// TIA Portal project "auto_level_palletizer_with_rotating_platform" (V15)

(* hardware
DEVICE "S7300/ET200M station_1"  S7-300 station
   slot 0: "Rail_0"  Rail  6ES7 390-1***0-0AA0
   slot 2: "controller_ALPwRP_system"  CPU 314C-2 PN/DP  6ES7 314-6EH04-0AB0  V3.3
      slot 2: "PROFINET interface_1"  PN-IO
         slot 1: "Port_1"  Port
         slot 2: "Port_2"  Port
      slot 5: "DI 24/DO 16_1"  DI24/DO16
      slot 6: "AI 5/AO 2_1"  AI5/AO2
      slot 7: "Count_1"  Counter
      slot 8: "Positioning_1"  Positioning
DEVICE "SINAMICS G_1"  Sinamics.Device
   slot 0: "CU240E-2 PN-F"  G120 CU240E-2 PN-F  6SL3244-0BB13-1FA0  4.7.9
      slot 1: "PROFINET interface"  MDD-SinamicsG120-P
   slot 0: "	_0"  Rail  SinamicsG120RackPN
   slot 3: "PM340 IP20"  PM340 IP20  6SL3210-1SB11-0AA0  -
*)

// ===== PLC "controller_ALPwRP_system"  CPU 314C-2 PN/DP =====

VAR_GLOBAL   // PLC tag table "Default tag table"
   "1B1" AT %I0.0 : Bool;   // Carton Passed
   "2B1" AT %I0.1 : Bool;   // Carton Counter
   "3B1" AT %I0.2 : Bool;   // Feeding Actuator 3A Fully Retracted
   "3B2" AT %I0.3 : Bool;   // Feeding Actuator 3A Fully Extended
   "3B3" AT %I0.4 : Bool;   // Feeding Actuator 3A in X position
   "4B1" AT %I0.5 : Bool;   // Sheet Motor 4A Fully Retracted
   "4B2" AT %I0.6 : Bool;   // Sheet Motor 4A Fully Extended
   "4B3" AT %I0.7 : Bool;   // Sheet Motor 4A in L position
   "5B1" AT %I1.0 : Bool;   // Carton to the feeding station
   "6B1" AT %I1.1 : Bool;   // Rotating Platform is ready (90 degrees)
   "7B1" AT %I1.2 : Bool;   // Hydraulic lift 6A Fully extended
   "7B2" AT %I1.3 : Bool;   // Hydraulic lift 6A Fully retracted
   "7B3" AT %I1.4 : Bool;   // Hydrauic Cylinder in Y
   "8B1" AT %I1.5 : Bool;   // Pallet Available
   "9B1" AT %I1.6 : Bool;   // Alignment Stopper 7A Fully Extended
   "9B2" AT %I1.7 : Bool;   // Alignment Stopper 7A Fully Retracted
   "10B1" AT %I2.0 : Bool;   // Carton to Alignment Actuator
   "S1" AT %I2.1 : Bool;   // START BUTTON PUSHED
   "S2" AT %I2.2 : Bool;   // STOP BUTTON PUSHED
   "S3" AT %I2.3 : Bool;   // RESET BUTTON PUSHED
   "EM_STOP" AT %I2.4 : Bool;   // EMERGENCY BUTTON PUSHED
   "11B1" AT %I2.5 : Bool;   // 8 AWG Carton Type
   "11B2" AT %I2.6 : Bool;   // 10 AWG Carton Type
   "11B3" AT %I2.7 : Bool;   // 12, 14, & 16 AWG Carton Types
   "M1" AT %Q0.0 : Bool;   // Belt Conveyor 1A
   "M2" AT %Q0.1 : Bool;   // Roller Conveyor 2A
   "M3" AT %Q0.2 : Bool;   // Feeding Actuator 3A
   "M4" AT %Q0.3 : Bool;   // Sheet Metal
   "P2" AT %Q0.4 : Bool;   // Pallet Rotation 5A
   "P1" AT %Q0.5 : Bool;   // Pallet z Axis 6A
   "A2" AT %Q0.6 : Bool;   // Aligment Stopper 7A
   "Tag_1" AT %M0.0 : Bool;
END_VAR

DATA_BLOCK "Main Program_DB"   // DB2
{ S7_Optimized_Access := 'FALSE' }
VERSION : 0.1
// stored: InstanceOfName Main Program
"Main Program"
BEGIN
END_DATA_BLOCK

FUNCTION_BLOCK "Main Program"   // FB1, GRAPH
{ S7_Optimized_Access := 'FALSE' }
VERSION : 0.1
   VAR_INPUT
      OFF_SQ : Bool := false;   // Turn sequence off
      INIT_SQ : Bool := false;   // Set sequence to initial state
      ACK_EF : Bool := false;   // Acknowledge all errors and faults
      S_PREV : Bool := false;   // Output previous step in parameter S_NO
      S_NEXT : Bool := false;   // Indicate next step in parameter S_NO
      SW_AUTO : Bool := false;   // Automatic mode
      SW_TAP : Bool := false;   // Semiautomatic/switch with transition
      SW_TOP : Bool := false;   // Semiautomatic/ignore transition
      SW_MAN : Bool := false;   // Manual mode
      S_SEL : Int := 0;   // Select step to be output to S_NO
      S_ON : Bool := false;   // Activate step indicated in S_NO
      S_OFF : Bool := false;   // Deactivate step indicated S_NO
      T_PUSH : Bool := false;   // Enable transition to switch in semi automatic mode
   END_VAR
   VAR_OUTPUT
      S_NO : Int := 0;   // Step number
      S_MORE : Bool := false;   // More steps are available and can be shown in S_NO
      S_ACTIVE : Bool := false;   // Step indicated in S_NO is active
      ERR_FLT : Bool := false;   // Interlock or supervision group error
      AUTO_ON : Bool := false;   // Automatic mode is active
      TAP_ON : Bool := false;   // Semiautomatic mode/step with transition enabled
      TOP_ON : Bool := false;   // Semiautomatic mode/ignore transition enabled
      MAN_ON : Bool := false;   // Manual mode is active
   END_VAR
   VAR
      in_initial_position : Bool;
      SWITCH : Array[0..0] of DWord;
      SW_SQTS : Array[0..21] of Byte;
      SW_ADDR : Word := 16#C;
      G7T_0 : GraphTransition;
      G7S_0 : GraphStep;
      PRE_CRIT : Array[0..0] of DWord;
      POST_CRIT : Array[0..0] of DWord;
      TVX : Array[0..5] of Byte;
      TTX : Array[0..5] of Byte;
      TSX : Array[0..2] of Byte;
      S00X : Array[0..2] of Byte;
      SOFFX : Array[0..2] of Byte;
      SONX : Array[0..2] of Byte;
      SAX : Array[0..2] of Byte;
      SERRX : Array[0..22] of Byte;
      SMX : Array[0..22] of Byte;
      S0X : Array[0..22] of Byte;
      S1X : Array[0..22] of Byte;
      S_DISPLAY : Int;   // Internal display of output parameter S_NO
      S_SEL_OLD : Int;   // Previous value in S_SEL
      S_DISPIDX : Byte;   // Index of the step in S_NO
      T_DISPIDX : Byte;   // Index of the transition displayed in T_NO
      MOPEDGE : Struct
         AUTO : Bool := false;
         MAN : Bool := false;
         TAP : Bool := false;
         TOP : Bool := false;
         ACK_S : Bool := false;
         REG_S : Bool := false;
         T_PREV : Bool := false;
         T_NEXT : Bool := false;
         LOCK : Bool := false;
         SUP : Bool := false;
         ACKREQ : Bool := false;
         SSKIP : Bool := false;
         OFF : Bool := false;
         INIT : Bool := false;
         HALT : Bool := false;
         TMS_HALT : Bool := false;
         OPS_ZERO : Bool := false;
         SACT_DISP : Bool := false;
         SEF_DISP : Bool := false;
         SALL_DISP : Bool := false;
         S_PREV : Bool := false;
         S_NEXT : Bool := false;
         S_SELOK : Bool := false;
         S_ON : Bool := false;
         S_OFF : Bool := false;
         T_PUSH : Bool := false;
         REG : Bool := false;
         ACK : Bool := false;
         IL_PERM : Bool := false;
         T_PERM : Bool := false;
         ILP_MAN : Bool := false;
      END_STRUCT;
      MOP : Struct   // Mode
         AUTO : Bool := true;   // Status: automatic mode
         MAN : Bool := false;   // Status: manual mode
         TAP : Bool := false;   // Status: semi automatic/switch with transition
         TOP : Bool := false;   // Status: semi automatic/ignore transition
         ACK_S : Bool := false;   // Request: acknowledge step at parameter S_NO
         REG_S : Bool := false;   // Request: register step indicated in S_NO
         T_PREV : Bool := false;   // Request: output previous valid transition in T_NO
         T_NEXT : Bool := false;   // Request: output next valid transition in T_NO
         LOCK : Bool := true;   // Status: interlocks activated
         SUP : Bool := true;   // Status: supervisions activated
         ACKREQ : Bool := true;   // Status: acknowledgment required
         SSKIP : Bool := false;   // Status: "Skip steps" enabled
         OFF : Bool := false;   // Request: deactivate all steps
         INIT : Bool := true;   // Request: set sequence to initial state
         HALT : Bool := false;   // Status: sequence halted
         TMS_HALT : Bool := false;   // Status: all internal timers held
         OPS_ZERO : Bool := false;   // Status: set all operands processed with N, L, D instructions to 0
         SACT_DISP : Bool := true;   // Status: display active steps only
         SEF_DISP : Bool := false;   // Status: display only steps with errors and disrupted steps
         SALL_DISP : Bool := false;   // Status: display all steps
         S_PREV : Bool := false;   // Request: output previous step to S_NO
         S_NEXT : Bool := false;   // Request: Output next step at S_NO parameter
         S_SELOK : Bool := false;   // Request: output step number from S_SEL to S_NO
         S_ON : Bool := false;   // Request: activate step indicated in S_NO
         S_OFF : Bool := false;   // Request: deactivate step at parameter S_NO
         T_PUSH : Bool := false;   // Request: transition switching enabled
         REG : Bool := false;   // Request: register all interlock and supervision errors
         ACK : Bool := false;   // Request: acknowledge all interlock and supervision errors
         IL_PERM : Bool := false;   // Status: permanent processing of all interlocks
         T_PERM : Bool := false;   // Status: permanent processing of all transitions
         ILP_MAN : Bool := false;   // Status: permanent processing of all interlocks in manual mode
      END_STRUCT;
      TICKS : Struct   // Clock speeds
         DELTA : Time := T#0ms;   // Time difference between cycles
         OLD : Time := T#0ms;   // 10 ms clock counter value in last cycle
         NEW : Time := T#0ms;   // 10 ms clock counter value in this cycle
      END_STRUCT;
      SQ_FLAGS : Struct   // Sequence bit memory
         ERR_FLT : Bool := false;   // Interlock and supervision group error
         ERROR : Bool := false;   // Interlock group error
         FAULT : Bool := false;   // Supervision group error
         RT_FAIL : Bool := false;   // Runtime error
         NO_SNO : Bool := false;   // Requested step number not found
         NF_OFL : Bool := false;   // Overflow: too many ON or OFF requests
         SA_OFL : Bool := false;   // Overflow: too many steps active
         TV_OFL : Bool := false;   // Overflow: too many valid transitions
         MSG_OFL : Bool := false;   // Overflow: not enough system resources for ALARM_S
         NO_SWI : Bool := false;   // Do not switch in this cycle
         CYC_OP : Bool := false;   // Cyclic execution of the sequence after initialization
         AS_MSG : Bool := true;   // Alarms during runtime enabled or disabled by instruction
         AS_SEND : Bool := false;   // Send alarms from WR_USMSG or only enter in diagnostics buffer
         SQ_BUSY : Bool := false;   // Internal edge memory bit for sequence processing
         SA_BUSY : Bool := false;   // Internal edge memory bit for sequence processing
         AS_SIG : Bool := false;   // Edge memory bit for alarms from Alarm_S and Alarm_SQ
      END_STRUCT;
      S_PTR : DWord := 16#D40;
      S_PTR2 : DWord := 16#0;
      S_PTR3 : DWord := 16#26C0;
      S_PTR4 : DWord := 16#2600;
      T_PTR : DWord := 16#2540;
      C_AR2 : DWord := 16#0;
      M_FBDB : DWord := 16#10000;
      M_SNO : Word := 16#1;
      M_EVID : Word := 16#0;
      M_EVIL : C_Alarm_s;
      M_EVSV : C_Alarm_s;
      M_EV : DWord := 16#2420;
      CRIT : Array[0..31] of Bool;
      S_START : Byte := 16#0;
      S_IDX : Byte := 16#0;
      S_INT : Int := 72;
      S_TMP : Byte := 16#0;
      T_START : Byte := 16#0;
      T_IDX : Byte := 16#0;
      T_TMP : Byte := 16#0;
      T_TMP2 : Byte := 16#00;
      TV_POT : Byte := 16#06;
      RETURN1 : Byte := 16#0;
      RETURN2 : Byte := 16#0;
      SINI : Array[0..2] of Byte;
      LSTT : Array[0..23] of Byte;
      ATAJ : Array[0..23] of Byte;
      ATAB : Array[0..23] of Byte;
      PSTT : Array[0..23] of Byte;
      NSTT : Array[0..23] of Byte;
      ASSJ : Array[0..21] of Byte;
      ASSB : Array[0..21] of Byte;
      PTTS : Array[0..21] of Byte;
      NTTS : Array[0..21] of Byte;
      PRE_CNT : Word := 16#1;
      POST_CNT : Word := 16#1;
      ADR_COND : Word := 16#0;
      MAX_TVAL : Byte := 16#4;
      MAX_SACT : Byte := 16#1;
      MAX_CRIT : Byte := 16#4;
      T_CNT : Byte := 16#17;
      SUP_CNT : Byte := 16#0;
      LOCK_CNT : Byte := 16#0;
      S_CNT : Byte := 16#15;
      SQ_CNT : Byte := 16#1;
      PRS_INPAR : DWord := 16#E000FEC8;
      PRS_OUTPAR : DWord := 16#E000800F;
      GC_FLAGS : Struct
         T_MACH : Byte := 16#EB;
         COND_ED : Byte := 16#E3;
         W_LEVEL : Byte := 16#D5;
         FB_IF : Byte := 16#FA;
         AS_MSG : Word := 16#404;
         SSB : Word := 16#108;
         DILG : Word := 16#644;
         ADDR_T0 : Word := 16#28;
         CRIT_AVAIL : Bool := false;
         SSKIP_AVAIL : Bool := true;
         SSKIP_ON : Bool := false;
         ACK_REQ : Bool := true;
         SYNC_AVAIL : Bool := true;
         ILP_MAN : Bool := false;
         SWM_LOCKED : Bool := false;
         SAVE_SW : Bool := true;
      END_STRUCT;
      G7_FBMARK : Byte := 16#3C;
      G7_RELEASE : Byte := 16#3C;
      G7_ID2 : Byte := 16#37;
      G7_ID1 : Byte := 16#47;
   END_VAR
   VAR_TEMP
      EoF1 : Bool;   // End of "place_cartons_on_pallet" Function
      EoF2 : Bool;   // End of "palletize_cartons_on_pallet" Function
   END_VAR
   VAR CONSTANT
      X0 : Real;   // Pushing Arm Retraction Position
      X1_8AWG : Real;   // Pushing Arm 8-AWG Odd Floors 1st carton
      X2_8AWG : Real;   // Pushing Arm 8-AWG Odd Floors 2nd carton.
      X3_8AWG : Real;   // Pushing Arm 8-AWG Holding cartons position (2)
      X4_8AWG : Real;   // Pushing Arm 8-AWG Even Floors 4-carton row
      X5_8AWG : Real;   // Pushing Arm Holding cartons position (4)
      L0 : Real;   // Sheet Metal Initial Position
      L1 : Real;   // Sheet Metal 8-AWG Midway Position
      L2 : Real;   // Sheet Metal Fully Extension Position
      Z4_8AWG : Real;   // 1st Carton-Floor Altitude
      Z3_8AWG : Real;   // 2nd Carton-Floor Altitude
      Z2_8AWG : Real;   // 3rd Carton-Floor Altitude
      Z1_8AWG : Real;   // 4th Carton-Floor Altitude
      Z0_8AWG : Real;   // Last Carton-Floor Altitude
      no_rotation : Int := 0;
      degree_90 : Int := 1;
      X1_10AWG : Real;   // 1st row position (3*4)
      X2_10AWG : Real;   // 2nd row position ( 3*4)
      X3_10AWG : Real;   // 3rd row position (3*4)
      X4_10AWG : Real;   // Floor stopping position
      X5_10AWG : Real;   // 1st row position (2*6)
      X6_10AWG : Real;   // 2nd row position (2*6)
      X7_10AWG : Real;   // Floor stopping position (2*6)
      Z5_10AWG : Real;   // 1st Carton-Floor Altitude
      Z4_10AWG : Real;   // 2nd Carton-Floor Altitude
      Z3_10AWG : Real;   // 3rd Carton-Floor Altitude
      Z2_10AWG : Real;   // 4th Carton-Floor Altitude
      Z1_10AWG : Real;   // 5th Carton-Floor Altitude
      Z0_10AWG : Real;   // Pallet is ready to move
      X1_12AWG : Real := 0.0;   // 1st row position (3*2)
      X2_12AWG : Real := 0.0;   // 2nd row position ( 3*2)
      X3_12AWG : Real := 0.0;   // Floor Stopping Position (3*2)
      Z6_12AWG : Real;   // 1st Floor Altitude
      Z5_12AWG : Real := 0.0;   // 2nd Floor Altitude
      Z4_12AWG : Real := 0.0;   // 3rd Floor Altitude
      Z3_12AWG : Real := 0.0;   // 4th Floor Altitude
      Z2_12AWG : Real := 0.0;   // 5th Floor Altitude
      Z1_12AWG : Real := 0.0;   // 6th Floor Altitude
      Z0_12AWG : Real := 0.0;   // Pallet is ready to move
   END_VAR
   // SW_SQTS[0] := 16#5;
   // SW_SQTS[3] := 16#1;
   // SW_SQTS[4] := 16#2;
   // SW_SQTS[5] := 16#3;
   // SW_SQTS[6] := 16#1;
   // SW_SQTS[7] := 16#1;
   // SW_SQTS[8] := 16#1;
   // SW_SQTS[9] := 16#1;
   // SW_SQTS[10] := 16#1;
   // SW_SQTS[11] := 16#2;
   // SW_SQTS[12] := 16#2;
   // SW_SQTS[13] := 16#2;
   // SW_SQTS[14] := 16#2;
   // SW_SQTS[15] := 16#2;
   // SW_SQTS[16] := 16#2;
   // SW_SQTS[17] := 16#2;
   // SW_SQTS[18] := 16#3;
   // SW_SQTS[19] := 16#3;
   // SW_SQTS[20] := 16#3;
   // SW_SQTS[21] := 16#4;
   // TVX[0] := 16#1;
   // TTX[0] := 16#1;
   // TSX[0] := 16#1;
   // S00X[0] := 16#1;
   // SOFFX[0] := 16#1;
   // SONX[0] := 16#1;
   // SAX[0] := 16#1;
   // SERRX[0] := 16#1;
   // SMX[0] := 16#1;
   // S0X[0] := 16#1;
   // S1X[0] := 16#1;
   // SINI[0] := 16#2;
   // SINI[1] := 16#1;
   // SINI[2] := 0;
   // LSTT[0] := 0;
   // LSTT[1] := 0;
   // LSTT[2] := 0;
   // LSTT[3] := 0;
   // LSTT[4] := 0;
   // LSTT[5] := 0;
   // LSTT[6] := 0;
   // LSTT[7] := 0;
   // LSTT[8] := 0;
   // LSTT[9] := 0;
   // LSTT[10] := 0;
   // LSTT[11] := 0;
   // LSTT[12] := 0;
   // LSTT[13] := 0;
   // LSTT[14] := 0;
   // LSTT[15] := 0;
   // LSTT[16] := 0;
   // LSTT[17] := 0;
   // LSTT[18] := 0;
   // LSTT[19] := 0;
   // LSTT[20] := 0;
   // LSTT[21] := 0;
   // LSTT[22] := 0;
   // LSTT[23] := 16#1;
   // ATAJ[0] := 0;
   // ATAJ[1] := 16#1;
   // ATAJ[2] := 16#2;
   // ATAJ[3] := 16#3;
   // ATAJ[4] := 16#4;
   // ATAJ[5] := 16#5;
   // ATAJ[6] := 16#6;
   // ATAJ[7] := 16#7;
   // ATAJ[8] := 16#8;
   // ATAJ[9] := 16#9;
   // ATAJ[10] := 16#A;
   // ATAJ[11] := 16#B;
   // ATAJ[12] := 16#13;
   // ATAJ[13] := 16#D;
   // ATAJ[14] := 16#E;
   // ATAJ[15] := 16#F;
   // ATAJ[16] := 16#10;
   // ATAJ[17] := 16#11;
   // ATAJ[18] := 16#12;
   // ATAJ[19] := 16#16;
   // ATAJ[20] := 16#14;
   // ATAJ[21] := 16#15;
   // ATAJ[22] := 16#C;
   // ATAJ[23] := 16#17;
   // ATAB[0] := 0;
   // ATAB[1] := 16#1;
   // ATAB[2] := 16#3;
   // ATAB[3] := 16#4;
   // ATAB[4] := 16#2;
   // ATAB[5] := 16#5;
   // ATAB[6] := 16#6;
   // ATAB[7] := 16#7;
   // ATAB[8] := 16#8;
   // ATAB[9] := 16#9;
   // ATAB[10] := 16#A;
   // ATAB[11] := 16#B;
   // ATAB[12] := 16#C;
   // ATAB[13] := 16#D;
   // ATAB[14] := 16#E;
   // ATAB[15] := 16#F;
   // ATAB[16] := 16#10;
   // ATAB[17] := 16#11;
   // ATAB[18] := 16#12;
   // ATAB[19] := 16#13;
   // ATAB[20] := 16#14;
   // ATAB[21] := 16#15;
   // ATAB[22] := 16#16;
   // ATAB[23] := 16#17;
   // PSTT[0] := 0;
   // PSTT[1] := 16#1;
   // PSTT[2] := 16#2;
   // PSTT[3] := 16#2;
   // PSTT[4] := 16#2;
   // PSTT[5] := 16#3;
   // PSTT[6] := 16#4;
   // PSTT[7] := 16#5;
   // PSTT[8] := 16#6;
   // PSTT[9] := 16#7;
   // PSTT[10] := 16#8;
   // PSTT[11] := 16#9;
   // PSTT[12] := 16#A;
   // PSTT[13] := 16#B;
   // PSTT[14] := 16#C;
   // PSTT[15] := 16#E;
   // PSTT[16] := 16#D;
   // PSTT[17] := 16#F;
   // PSTT[18] := 16#10;
   // PSTT[19] := 16#11;
   // PSTT[20] := 16#12;
   // PSTT[21] := 16#13;
   // PSTT[22] := 16#14;
   // PSTT[23] := 16#15;
   // NSTT[0] := 16#1;
   // NSTT[1] := 16#2;
   // NSTT[2] := 16#4;
   // NSTT[3] := 16#5;
   // NSTT[4] := 16#3;
   // NSTT[5] := 16#6;
   // NSTT[6] := 16#B;
   // NSTT[7] := 16#12;
   // NSTT[8] := 16#7;
   // NSTT[9] := 16#8;
   // NSTT[10] := 16#9;
   // NSTT[11] := 16#A;
   // NSTT[12] := 16#15;
   // NSTT[13] := 16#C;
   // NSTT[14] := 16#D;
   // NSTT[15] := 16#F;
   // NSTT[16] := 16#E;
   // NSTT[17] := 16#10;
   // NSTT[18] := 16#11;
   // NSTT[19] := 16#15;
   // NSTT[20] := 16#13;
   // NSTT[21] := 16#14;
   // NSTT[22] := 16#15;
   // NSTT[23] := 16#1;
   // ASSJ[0] := 0;
   // ASSJ[1] := 16#1;
   // ASSJ[2] := 16#2;
   // ASSJ[3] := 16#3;
   // ASSJ[4] := 16#4;
   // ASSJ[5] := 16#5;
   // ASSJ[6] := 16#6;
   // ASSJ[7] := 16#7;
   // ASSJ[8] := 16#8;
   // ASSJ[9] := 16#9;
   // ASSJ[10] := 16#A;
   // ASSJ[11] := 16#B;
   // ASSJ[12] := 16#C;
   // ASSJ[13] := 16#D;
   // ASSJ[14] := 16#E;
   // ASSJ[15] := 16#F;
   // ASSJ[16] := 16#10;
   // ASSJ[17] := 16#11;
   // ASSJ[18] := 16#12;
   // ASSJ[19] := 16#13;
   // ASSJ[20] := 16#14;
   // ASSJ[21] := 16#15;
   // ASSB[0] := 0;
   // ASSB[1] := 16#1;
   // ASSB[2] := 16#2;
   // ASSB[3] := 16#3;
   // ASSB[4] := 16#4;
   // ASSB[5] := 16#5;
   // ASSB[6] := 16#6;
   // ASSB[7] := 16#7;
   // ASSB[8] := 16#8;
   // ASSB[9] := 16#9;
   // ASSB[10] := 16#A;
   // ASSB[11] := 16#B;
   // ASSB[12] := 16#C;
   // ASSB[13] := 16#D;
   // ASSB[14] := 16#E;
   // ASSB[15] := 16#F;
   // ASSB[16] := 16#10;
   // ASSB[17] := 16#11;
   // ASSB[18] := 16#12;
   // ASSB[19] := 16#13;
   // ASSB[20] := 16#14;
   // ASSB[21] := 16#15;
   // PTTS[0] := 0;
   // PTTS[2] := 16#1;
   // PTTS[3] := 16#4;
   // PTTS[4] := 16#2;
   // PTTS[5] := 16#3;
   // PTTS[6] := 16#5;
   // PTTS[7] := 16#8;
   // PTTS[8] := 16#9;
   // PTTS[9] := 16#A;
   // PTTS[10] := 16#B;
   // PTTS[11] := 16#6;
   // PTTS[12] := 16#D;
   // PTTS[13] := 16#E;
   // PTTS[14] := 16#10;
   // PTTS[15] := 16#F;
   // PTTS[16] := 16#11;
   // PTTS[17] := 16#12;
   // PTTS[18] := 16#7;
   // PTTS[19] := 16#14;
   // PTTS[20] := 16#15;
   // PTTS[21] := 16#C;
   // NTTS[0] := 0;
   // NTTS[1] := 16#1;
   // NTTS[2] := 16#4;
   // NTTS[3] := 16#5;
   // NTTS[4] := 16#6;
   // NTTS[5] := 16#7;
   // NTTS[6] := 16#8;
   // NTTS[7] := 16#9;
   // NTTS[8] := 16#A;
   // NTTS[9] := 16#B;
   // NTTS[10] := 16#C;
   // NTTS[11] := 16#D;
   // NTTS[12] := 16#E;
   // NTTS[13] := 16#10;
   // NTTS[14] := 16#F;
   // NTTS[15] := 16#11;
   // NTTS[16] := 16#12;
   // NTTS[17] := 16#13;
   // NTTS[18] := 16#14;
   // NTTS[19] := 16#15;
   // NTTS[20] := 16#16;
   // NTTS[21] := 16#17;
BEGIN
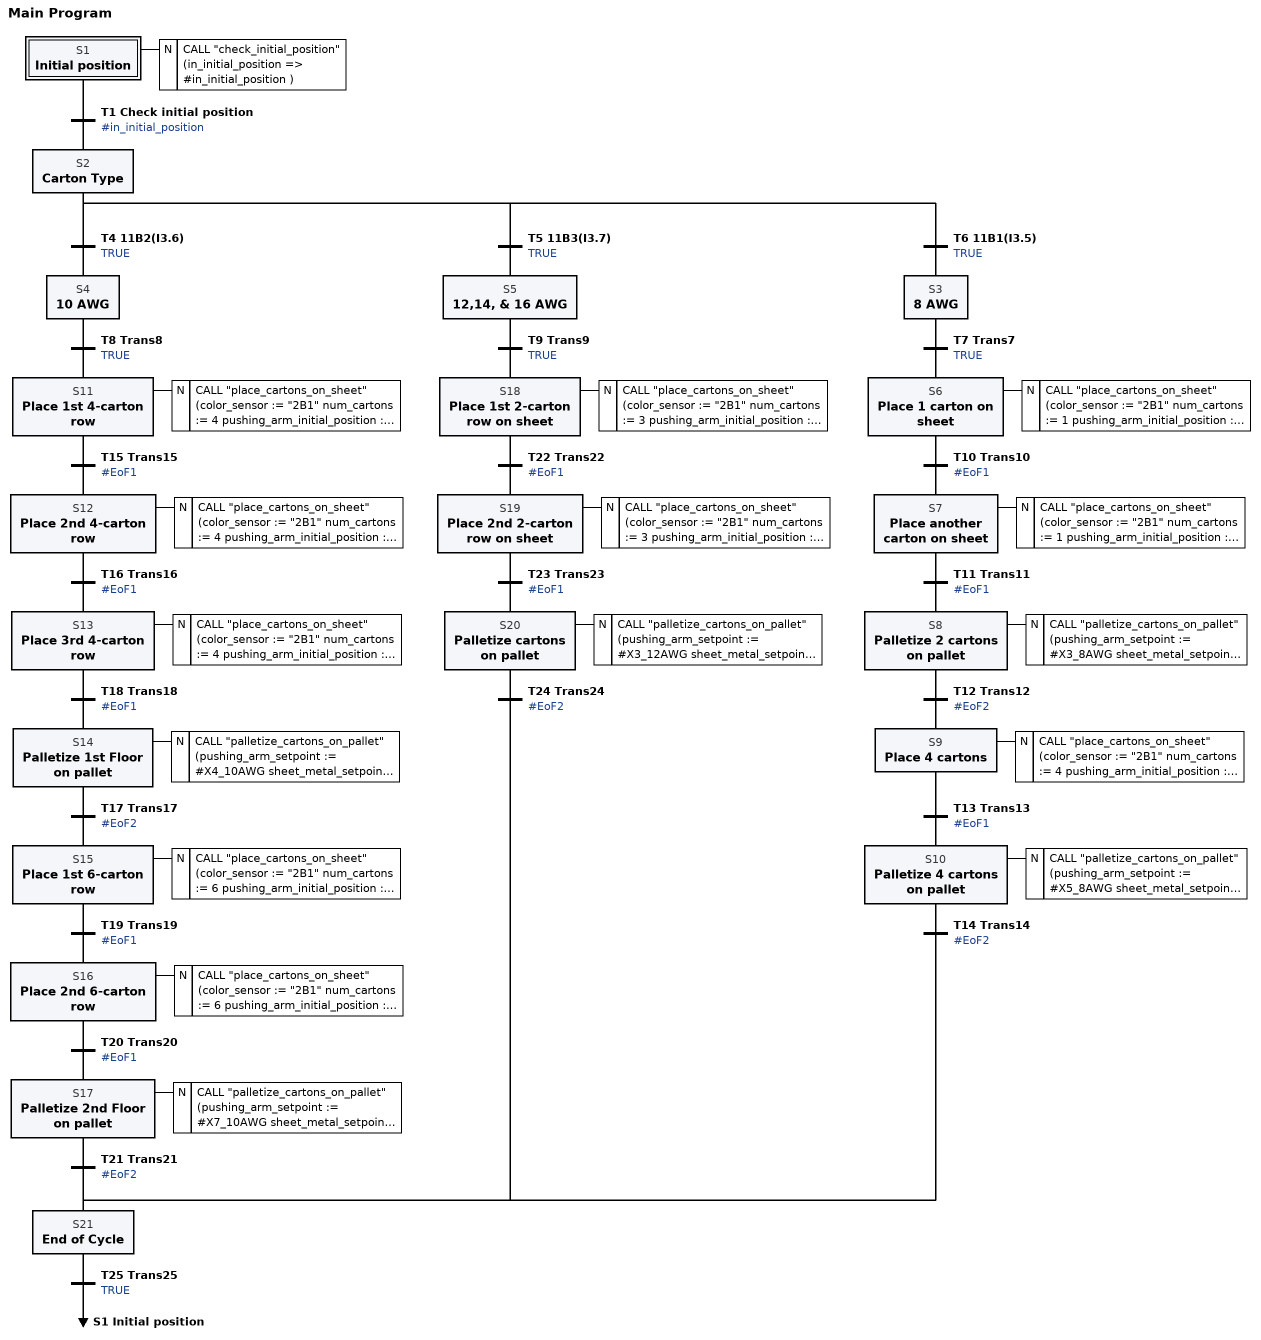
   // sequencer 1
   INITIAL_STEP "Initial position":   // S1
              N    CALL "check_initial_position"
                   (in_initial_position => #in_initial_position
                   )
   END_STEP
   TRANSITION "Check initial position" FROM "Initial position" TO "Carton Type"   // T1
      := #in_initial_position;
   END_TRANSITION
   STEP "Carton Type":   // S2
   END_STEP
   TRANSITION "11B2(I3.6)" FROM "Carton Type" TO "10 AWG"   // T4
      := TRUE;
   END_TRANSITION
   TRANSITION "11B3(I3.7)" FROM "Carton Type" TO "12,14, & 16 AWG"   // T5
      := TRUE;
   END_TRANSITION
   TRANSITION "11B1(I3.5)" FROM "Carton Type" TO "8 AWG"   // T6
      := TRUE;
   END_TRANSITION
   STEP "8 AWG":   // S3
   END_STEP
   TRANSITION Trans7 FROM "8 AWG" TO "Place 1 carton on sheet"   // T7
      := TRUE;
   END_TRANSITION
   STEP "10 AWG":   // S4
   END_STEP
   TRANSITION Trans8 FROM "10 AWG" TO "Place 1st 4-carton row"   // T8
      := TRUE;
   END_TRANSITION
   STEP "12,14, & 16 AWG":   // S5
   END_STEP
   TRANSITION Trans9 FROM "12,14, & 16 AWG" TO "Place 1st 2-carton row on sheet"   // T9
      := TRUE;
   END_TRANSITION
   STEP "Place 1 carton on sheet":   // S6
              N    CALL "place_cartons_on_sheet"
                   (color_sensor := "2B1"
                   num_cartons := 1
                   pushing_arm_initial_position := #X0
                   pushing_arm_setpoint := #X1_8AWG
                   retract_arm := True
                   alignment := True
                   EoF => #EoF1
                   )
   END_STEP
   TRANSITION Trans10 FROM "Place 1 carton on sheet" TO "Place another carton on sheet"   // T10
      := #EoF1;
   END_TRANSITION
   STEP "Place another carton on sheet":   // S7
              N    CALL "place_cartons_on_sheet"
                   (color_sensor := "2B1"
                   num_cartons := 1
                   pushing_arm_initial_position := #X0
                   pushing_arm_setpoint := #X2_8AWG
                   retract_arm := 0
                   alignment := 1
                   EoF => #EoF1
                   )
   END_STEP
   TRANSITION Trans11 FROM "Place another carton on sheet" TO "Palletize 2 cartons on pallet"   // T11
      := #EoF1;
   END_TRANSITION
   STEP "Palletize 2 cartons on pallet":   // S8
              N    CALL "palletize_cartons_on_pallet"
                   (pushing_arm_setpoint := #X3_8AWG
                   sheet_metal_setpoint := #L1
                   rotation_degree := #degree_90
                   EoF => #EoF2
                   )
   END_STEP
   TRANSITION Trans12 FROM "Palletize 2 cartons on pallet" TO "Place 4 cartons"   // T12
      := #EoF2;
   END_TRANSITION
   STEP "Place 4 cartons":   // S9
              N    CALL "place_cartons_on_sheet"
                   (color_sensor := "2B1"
                   num_cartons := 4
                   pushing_arm_initial_position := #X0
                   pushing_arm_setpoint := #X4_8AWG
                   retract_arm := 0
                   alignment := 0
                   EoF => #EoF1
                   )
   END_STEP
   TRANSITION Trans13 FROM "Place 4 cartons" TO "Palletize 4 cartons on pallet"   // T13
      := #EoF1;
   END_TRANSITION
   STEP "Palletize 4 cartons on pallet":   // S10
              N    CALL "palletize_cartons_on_pallet"
                   (pushing_arm_setpoint := #X5_8AWG
                   sheet_metal_setpoint := #L2
                   rotation_degree := #degree_90
                   EoF => #EoF2
                   )
   END_STEP
   TRANSITION Trans14 FROM "Palletize 4 cartons on pallet" TO "End of Cycle"   // T14
      := #EoF2;
   END_TRANSITION
   STEP "Place 1st 4-carton row":   // S11
              N    CALL "place_cartons_on_sheet"
                   (color_sensor := "2B1"
                   num_cartons := 4
                   pushing_arm_initial_position := #X0
                   pushing_arm_setpoint := #X1_10AWG
                   retract_arm := 1
                   alignment := 1
                   EoF => #EoF1
                   )
   END_STEP
   TRANSITION Trans15 FROM "Place 1st 4-carton row" TO "Place 2nd 4-carton row"   // T15
      := #EoF1;
   END_TRANSITION
   STEP "Place 2nd 4-carton row":   // S12
              N    CALL "place_cartons_on_sheet"
                   (color_sensor := "2B1"
                   num_cartons := 4
                   pushing_arm_initial_position := #X0
                   pushing_arm_setpoint := #X2_10AWG
                   retract_arm := 1
                   alignment := 1
                   EoF => #EoF1
                   )
   END_STEP
   TRANSITION Trans16 FROM "Place 2nd 4-carton row" TO "Place 3rd 4-carton row"   // T16
      := #EoF1;
   END_TRANSITION
   STEP "Place 3rd 4-carton row":   // S13
              N    CALL "place_cartons_on_sheet"
                   (color_sensor := "2B1"
                   num_cartons := 4
                   pushing_arm_initial_position := #X0
                   pushing_arm_setpoint := #X3_10AWG
                   retract_arm := 1
                   alignment := 1
                   EoF => #EoF1
                   )
   END_STEP
   TRANSITION Trans18 FROM "Place 3rd 4-carton row" TO "Palletize 1st Floor on pallet"   // T18
      := #EoF1;
   END_TRANSITION
   STEP "Palletize 1st Floor on pallet":   // S14
              N    CALL "palletize_cartons_on_pallet"
                   (pushing_arm_setpoint := #X4_10AWG
                   sheet_metal_setpoint := #L2
                   rotation_degree := #degree_90
                   EoF => #EoF2
                   )
   END_STEP
   TRANSITION Trans17 FROM "Palletize 1st Floor on pallet" TO "Place 1st 6-carton row"   // T17
      := #EoF2;
   END_TRANSITION
   STEP "Place 1st 6-carton row":   // S15
              N    CALL "place_cartons_on_sheet"
                   (color_sensor := "2B1"
                   num_cartons := 6
                   pushing_arm_initial_position := #X0
                   pushing_arm_setpoint := #X5_10AWG
                   retract_arm := 1
                   alignment := 0
                   EoF => #EoF1
                   )
   END_STEP
   TRANSITION Trans19 FROM "Place 1st 6-carton row" TO "Place 2nd 6-carton row"   // T19
      := #EoF1;
   END_TRANSITION
   STEP "Place 2nd 6-carton row":   // S16
              N    CALL "place_cartons_on_sheet"
                   (color_sensor := "2B1"
                   num_cartons := 6
                   pushing_arm_initial_position := #X0
                   pushing_arm_setpoint := #X6_10AWG
                   retract_arm := 1
                   alignment := 0
                   EoF => #EoF1
                   )
   END_STEP
   TRANSITION Trans20 FROM "Place 2nd 6-carton row" TO "Palletize 2nd Floor on pallet"   // T20
      := #EoF1;
   END_TRANSITION
   STEP "Palletize 2nd Floor on pallet":   // S17
              N    CALL "palletize_cartons_on_pallet"
                   (pushing_arm_setpoint := #X7_10AWG
                   sheet_metal_setpoint := #L2
                   rotation_degree := #degree_90
                   EoF => #EoF2
                   )
   END_STEP
   TRANSITION Trans21 FROM "Palletize 2nd Floor on pallet" TO "End of Cycle"   // T21
      := #EoF2;
   END_TRANSITION
   STEP "Place 1st 2-carton row on sheet":   // S18
              N    CALL "place_cartons_on_sheet"
                   (color_sensor := "2B1"
                   num_cartons := 3
                   pushing_arm_initial_position := #X0
                   pushing_arm_setpoint := #X1_12AWG
                   retract_arm := 1
                   alignment := 0
                   EoF => #EoF1
                   )
   END_STEP
   TRANSITION Trans22 FROM "Place 1st 2-carton row on sheet" TO "Place 2nd 2-carton row on sheet"   // T22
      := #EoF1;
   END_TRANSITION
   STEP "Place 2nd 2-carton row on sheet":   // S19
              N    CALL "place_cartons_on_sheet"
                   (color_sensor := "2B1"
                   num_cartons := 3
                   pushing_arm_initial_position := #X0
                   pushing_arm_setpoint := #X2_12AWG
                   retract_arm := 1
                   alignment := 0
                   EoF => #EoF1
                   )
   END_STEP
   TRANSITION Trans23 FROM "Place 2nd 2-carton row on sheet" TO "Palletize cartons on pallet"   // T23
      := #EoF1;
   END_TRANSITION
   STEP "Palletize cartons on pallet":   // S20
              N    CALL "palletize_cartons_on_pallet"
                   (pushing_arm_setpoint := #X3_12AWG
                   sheet_metal_setpoint := #L1
                   rotation_degree := 0
                   EoF => #EoF2
                   )
   END_STEP
   TRANSITION Trans24 FROM "Palletize cartons on pallet" TO "End of Cycle"   // T24
      := #EoF2;
   END_TRANSITION
   STEP "End of Cycle":   // S21
   END_STEP
   TRANSITION Trans25 FROM "End of Cycle" TO "Initial position"   // T25, jump
      := TRUE;
   END_TRANSITION
END_FUNCTION_BLOCK

FUNCTION "system_01" : Void   // FC1, LAD
{ S7_Optimized_Access := 'FALSE' }
VERSION : 0.1
   VAR_INPUT
      color_sensor : Bool;   // Signal color sensor
      reset_counter : Bool;   // Signal reset counter
      num_cartons : Int;   // Number of cartons to be placed on the sheet metal.
      x1 : Real;   // 1st positon setpoint for the pushing arm
      x2 : Real;   // 2nd position setpoint for the pushing arm
      is_aligned : Bool;   // Signal select alignment mode.
   END_VAR
   VAR_TEMP
      last_carton_passed : Bool;   // Last carton is counted or not
   END_VAR
   VAR CONSTANT
      motor_velocity : Real;
      motor_acceleration : Real;
      motor_deceleration : Real;
      motor_direction : Int;
   END_VAR
BEGIN

REGION Network 1: Roller Conveyor
   // Turn on the roller conveyor all the time.
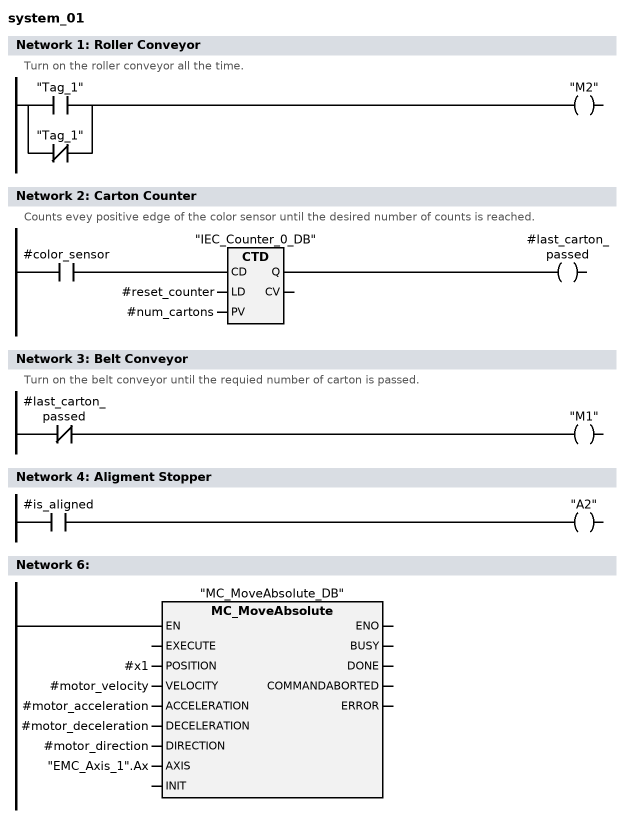
   RUNG wire#powerrail
      Contact( "Tag_1" )
      wire#w1
      Coil( "M2" )
   END_RUNG
   RUNG wire#powerrail
      I_Contact( "Tag_1" )
   END_RUNG wire#w1
   // the same network as SCL:
   "M2" := "Tag_1" OR NOT "Tag_1";
END_REGION

REGION Network 2: Carton Counter
   // Counts evey positive edge of the color sensor until the desired number of counts is reached.
   "IEC_Counter_0_DB".CTD(CD := #color_sensor, LD := #reset_counter, PV := #num_cartons);
   #last_carton_passed := "IEC_Counter_0_DB".Q;
END_REGION

REGION Network 3: Belt Conveyor
   // Turn on the belt conveyor until the requied number of carton is passed.
   RUNG wire#powerrail
      I_Contact( #last_carton_passed )
      Coil( "M1" )
   END_RUNG
   // the same network as SCL:
   "M1" := NOT #last_carton_passed;
END_REGION

REGION Network 4: Aligment Stopper
   RUNG wire#powerrail
      Contact( #is_aligned )
      Coil( "A2" )
   END_RUNG
   // the same network as SCL:
   "A2" := #is_aligned;
END_REGION

REGION Network 6
   "MC_MoveAbsolute_DB"(Position := #x1,   // MC_MoveAbsolute
                        Velocity := #motor_velocity,
                        Acceleration := #motor_acceleration,
                        Deceleration := #motor_deceleration,
                        Direction := #motor_direction,
                        Axis := "EMC_Axis_1".Ax);
END_REGION
END_FUNCTION

FUNCTION "place_cartons_on_sheet" : Void   // FC2, LAD
{ S7_Optimized_Access := 'FALSE' }
VERSION : 0.1
   VAR_INPUT
      color_sensor : Bool;   // Color sensor signal that decrements the counter with every positive edge.
      num_cartons : Int;   // Number of cartons required to be placed on the sheet.
      pushing_arm_initial_position : Real;   // Initial position for the pushing arm
      pushing_arm_setpoint : Real;   // Position setpoint for the pushing arm
      retract_arm : Bool;   // Determine whether the the pushing arm should return to its initial position.
      alignment : Bool;   // Determine whether the alignment should fully extend.
   END_VAR
   VAR_OUTPUT
      EoF : Bool;   // Indicate that all the required processes for this function has been carried out.
   END_VAR
   VAR_TEMP
      Last_carton_passed : Bool;   // Determine that the required numer of cartons has passed from the counter.
      Pushing_arm_in_position : Bool;   // Indicate that the pushing arm has reached its designated position and place the cartons on the sheet.
      cartons_ready : Bool;   // All the cartons arrived and are ready to be palltized by the pushing arm.
      Pushing_arm_is_retracted : Bool;   // Indicate whether the pushing arm is retracted after it places the carton on the sheet.
   END_VAR
   VAR CONSTANT
      waiting_time : Time := T#4MS;
      motor_velocity : Real;
      motor_acceleration : Real;
      motor_deceleration : Real;
      motor_direction : Int;
   END_VAR
BEGIN

REGION Network 1: Carton Couner Setup
   // Every positive edge of the color sensor signal will decrements the counter by one until it reaches zero. It will then return at the output "1", indicating that the required number of cartons have passed.
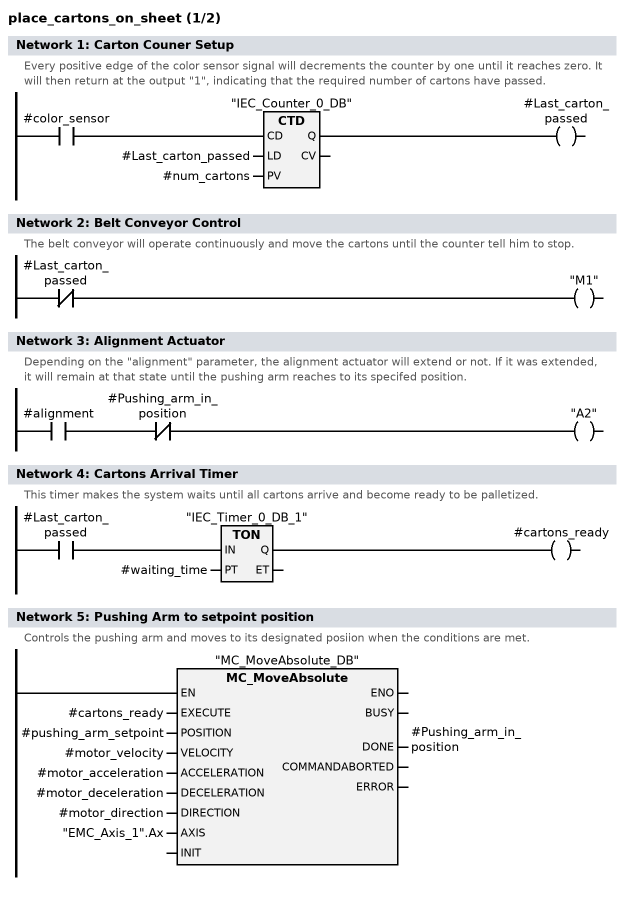
   "IEC_Counter_0_DB".CTD(CD := #color_sensor, LD := #Last_carton_passed, PV := #num_cartons);
   #Last_carton_passed := "IEC_Counter_0_DB".Q;
END_REGION

REGION Network 2: Belt Conveyor Control
   // The belt conveyor will operate continuously and move the cartons until the counter tell him to stop.
   RUNG wire#powerrail
      I_Contact( #Last_carton_passed )
      Coil( "M1" )
   END_RUNG
   // the same network as SCL:
   "M1" := NOT #Last_carton_passed;
END_REGION

REGION Network 3: Alignment Actuator
   // Depending on the "alignment" parameter, the alignment actuator will extend or not. If it was extended, it will remain at that state until the pushing arm reaches to its specifed position.
   RUNG wire#powerrail
      Contact( #alignment )
      I_Contact( #Pushing_arm_in_position )
      Coil( "A2" )
   END_RUNG
   // the same network as SCL:
   "A2" := #alignment AND NOT #Pushing_arm_in_position;
END_REGION

REGION Network 4: Cartons Arrival Timer
   // This timer makes the system waits until all cartons arrive and become ready to be palletized.
   "IEC_Timer_0_DB_1".TON(IN := #Last_carton_passed, PT := #waiting_time);
   #cartons_ready := "IEC_Timer_0_DB_1".Q;
END_REGION

REGION Network 5: Pushing Arm to setpoint position
   // Controls the pushing arm and moves to its designated posiion when the conditions are met.
   "MC_MoveAbsolute_DB"(Execute := #cartons_ready,   // MC_MoveAbsolute
                        Position := #pushing_arm_setpoint,
                        Velocity := #motor_velocity,
                        Acceleration := #motor_acceleration,
                        Deceleration := #motor_deceleration,
                        Direction := #motor_direction,
                        Axis := "EMC_Axis_1".Ax,
                        Done => #Pushing_arm_in_position);
END_REGION

REGION Network 6: Pushing Arm returns to its initial position.
   // Make the pushing arm returns to its initial position if that is required.
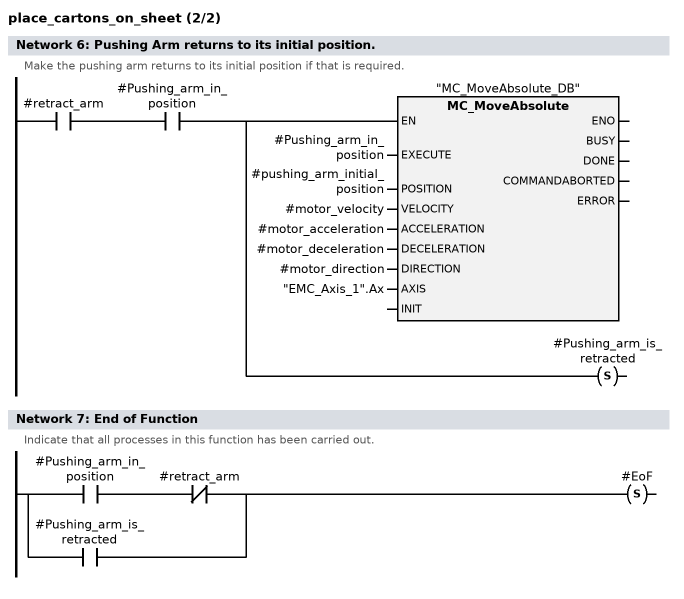
   IF #retract_arm AND #Pushing_arm_in_position THEN
       "MC_MoveAbsolute_DB"(Execute := #Pushing_arm_in_position,   // MC_MoveAbsolute
                            Position := #pushing_arm_initial_position,
                            Velocity := #motor_velocity,
                            Acceleration := #motor_acceleration,
                            Deceleration := #motor_deceleration,
                            Direction := #motor_direction,
                            Axis := "EMC_Axis_1".Ax);
       #Pushing_arm_is_retracted := TRUE;
   END_IF;
END_REGION

REGION Network 7: End of Function
   // Indicate that all processes in this function has been carried out.
   RUNG wire#powerrail
      Contact( #Pushing_arm_in_position )
      I_Contact( #retract_arm )
      wire#w1
      S_Coil( #EoF )
   END_RUNG
   RUNG wire#powerrail
      Contact( #Pushing_arm_is_retracted )
   END_RUNG wire#w1
   // the same network as SCL:
   IF (#Pushing_arm_in_position AND NOT #retract_arm) OR #Pushing_arm_is_retracted THEN #EoF := TRUE; END_IF;
END_REGION
END_FUNCTION

FUNCTION "palletize_cartons_on_pallet" : Void   // FC3, LAD
{ S7_Optimized_Access := 'FALSE' }
VERSION : 0.1
   VAR_INPUT
      pushing_arm_setpoint : Real;   // The position setpoint for the pushing arm.
      sheet_metal_setpoint : Real;   // The position setpoint for the sheet metak.
      rotation_degree : Int;   // The rotatiion degree for the rotating platform.
   END_VAR
   VAR_OUTPUT
      EoF : Bool;   // Indicates that all the required processes in this function has been carried out.
   END_VAR
   VAR_TEMP
      pushing_arm_in_position : Bool;   // Activates when the pushing arm reaches its designated position
      sheet_metal_in_positon : Bool;   // Activates when the sheet metal reaches its designated position
      do_it_once : Bool;
   END_VAR
   VAR CONSTANT
      pa_velocity : Real;   // Pushing arm's motor velocity
      pa_acceleration : Real;   // Pushig arm's motor acceleration
      pa_deceleration : Real;   // Pushing arm's motor deceleration
      pa_direction : Int;   // Pushing arm's motor direction
      sm_velocity : Real;   // Sheet metal's motor velocity
      sm_acceleration : Real;   // Sheet metal's motor acceleration
      sm_deceleration : Real;   // Sheet metal's motor deceleartion
      sm_direction : Int;   // Sheet metal's motor direction
      pushing_arm_initial_position : Real;   // Initial position for the pushing arm.
      sheet_metal_initial_position : Real;   // Initial position for the sheet metal.
   END_VAR
BEGIN

REGION Network 1: Sheet Metal to its designated position
   // Controls Sheet Metal and moves it to its designated position.
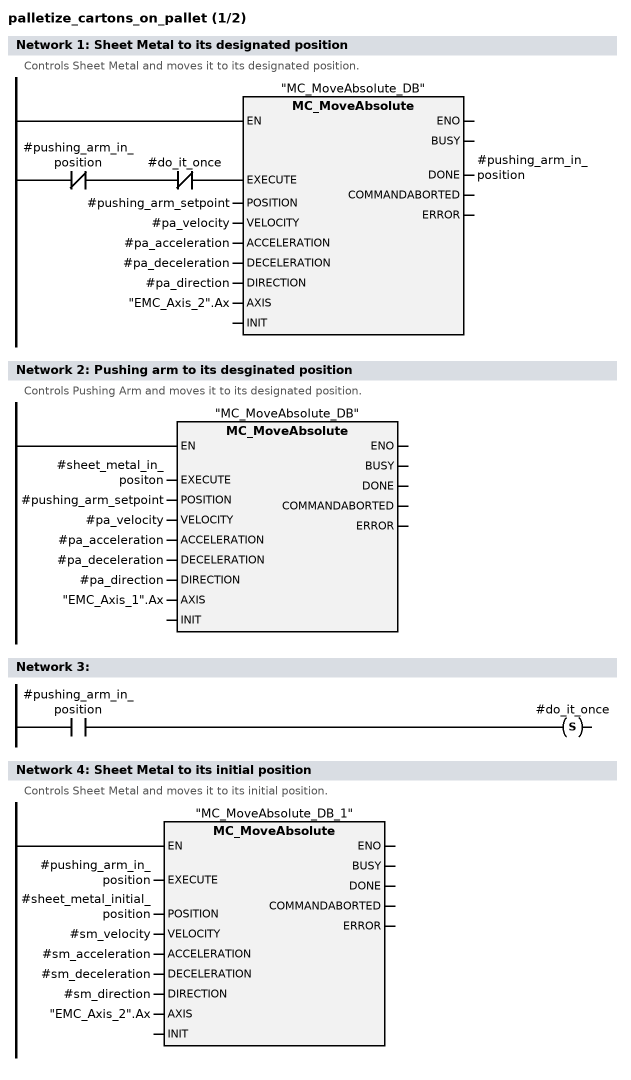
   "MC_MoveAbsolute_DB"(Execute := NOT #pushing_arm_in_position AND NOT #do_it_once,   // MC_MoveAbsolute
                        Position := #pushing_arm_setpoint,
                        Velocity := #pa_velocity,
                        Acceleration := #pa_acceleration,
                        Deceleration := #pa_deceleration,
                        Direction := #pa_direction,
                        Axis := "EMC_Axis_2".Ax,
                        Done => #pushing_arm_in_position);
END_REGION

REGION Network 2: Pushing arm to its desginated position
   // Controls Pushing Arm and moves it to its designated position.
   "MC_MoveAbsolute_DB"(Execute := #sheet_metal_in_positon,   // MC_MoveAbsolute
                        Position := #pushing_arm_setpoint,
                        Velocity := #pa_velocity,
                        Acceleration := #pa_acceleration,
                        Deceleration := #pa_deceleration,
                        Direction := #pa_direction,
                        Axis := "EMC_Axis_1".Ax);
END_REGION

REGION Network 3
   RUNG wire#powerrail
      Contact( #pushing_arm_in_position )
      S_Coil( #do_it_once )
   END_RUNG
   // the same network as SCL:
   IF #pushing_arm_in_position THEN #do_it_once := TRUE; END_IF;
END_REGION

REGION Network 4: Sheet Metal to its initial position
   // Controls Sheet Metal and moves it to its initial position.
   "MC_MoveAbsolute_DB_1"(Execute := #pushing_arm_in_position,   // MC_MoveAbsolute
                          Position := #sheet_metal_initial_position,
                          Velocity := #sm_velocity,
                          Acceleration := #sm_acceleration,
                          Deceleration := #sm_deceleration,
                          Direction := #sm_direction,
                          Axis := "EMC_Axis_2".Ax);
END_REGION

REGION Network 5: Pushing arm to its initial position
   // Controls Pushing Arm and moves it to its initial position.
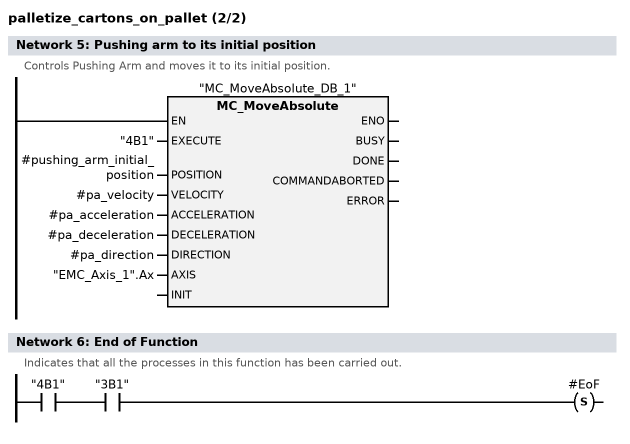
   "MC_MoveAbsolute_DB_1"(Execute := "4B1",   // MC_MoveAbsolute
                          Position := #pushing_arm_initial_position,
                          Velocity := #pa_velocity,
                          Acceleration := #pa_acceleration,
                          Deceleration := #pa_deceleration,
                          Direction := #pa_direction,
                          Axis := "EMC_Axis_1".Ax);
END_REGION

REGION Network 6: End of Function
   // Indicates that all the processes in this function has been carried out.
   RUNG wire#powerrail
      Contact( "4B1" )
      Contact( "3B1" )
      S_Coil( #EoF )
   END_RUNG
   // the same network as SCL:
   IF "4B1" AND "3B1" THEN #EoF := TRUE; END_IF;
END_REGION
END_FUNCTION

FUNCTION "check_initial_position" : Void   // FC4, LAD
{ S7_Optimized_Access := 'FALSE' }
VERSION : 0.1
   VAR_OUTPUT
      in_initial_position : Bool;
   END_VAR
BEGIN

REGION Network 1: Initial Position State
   // Check wether the system is in initial position or not.
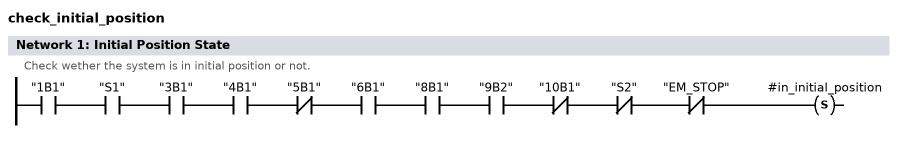
   RUNG wire#powerrail
      Contact( "1B1" )
      Contact( "S1" )
      Contact( "3B1" )
      Contact( "4B1" )
      I_Contact( "5B1" )
      Contact( "6B1" )
      Contact( "8B1" )
      Contact( "9B2" )
      I_Contact( "10B1" )
      I_Contact( "S2" )
      I_Contact( "EM_STOP" )
      S_Coil( #in_initial_position )
   END_RUNG
   // the same network as SCL:
   IF "1B1" AND "S1" AND "3B1" AND "4B1" AND NOT "5B1" AND "6B1" AND "8B1" AND "9B2" AND NOT "10B1" AND NOT "S2" AND NOT "EM_STOP" THEN
       #in_initial_position := TRUE;
   END_IF;
END_REGION
END_FUNCTION

ORGANIZATION_BLOCK "Main"   // OB1, LAD
TITLE = "Main Program Sweep (Cycle)"
{ S7_Optimized_Access := 'FALSE' }
VERSION : 0.1
   VAR_TEMP
      OB1_EV_CLASS : Byte;   // Bits 0-3 = 1 (Coming event), Bits 4-7 = 1 (Event class 1)
      OB1_SCAN_1 : Byte;   // 1 (Cold restart scan 1 of OB 1), 3 (Scan 2-n of OB 1)
      OB1_PRIORITY : Byte;   // Priority of OB Execution
      OB1_OB_NUMBR : Byte;   // 1 (Organization block 1, OB1)
      OB1_RESERVED_1 : Byte;   // Reserved for system
      OB1_RESERVED_2 : Byte;   // Reserved for system
      OB1_PREV_CYCLE : Int;   // Cycle time of previous OB1 scan (milliseconds)
      OB1_MIN_CYCLE : Int;   // Minimum cycle time of OB1 (milliseconds)
      OB1_MAX_CYCLE : Int;   // Maximum cycle time of OB1 (milliseconds)
      OB1_DATE_TIME : Date_And_Time;   // Date and time OB1 started
   END_VAR
BEGIN

REGION Network 1
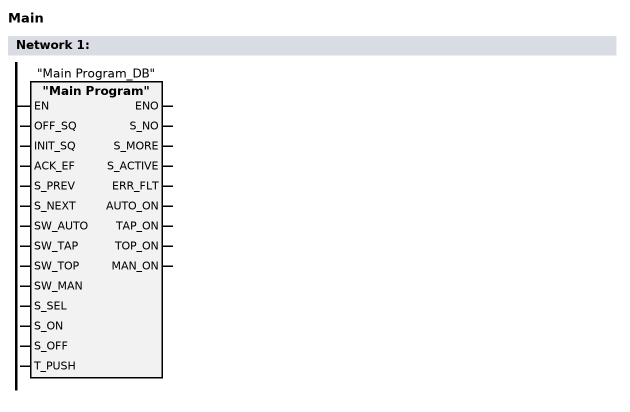
   RUNG wire#powerrail
      "Main Program_DB"(OFF_SQ :=, INIT_SQ :=, ACK_EF :=, S_PREV :=, S_NEXT :=, SW_AUTO :=, SW_TAP :=, SW_TOP :=, SW_MAN :=, S_SEL :=, S_ON :=, S_OFF :=, T_PUSH :=, S_NO =>, S_MORE =>, S_ACTIVE =>, ERR_FLT =>, AUTO_ON =>, TAP_ON =>, TOP_ON =>, MAN_ON =>)
   END_RUNG
   // the same network as SCL:
   "Main Program_DB"();   // "Main Program"
END_REGION
END_ORGANIZATION_BLOCK